// TIA Portal V15.1 export
// export: Created 2024-05-17T05:38:27.6005423Z, ExportSetting WithDefaults, DisplayName Totally Integrated Automation Portal, DisplayVersion V15.1 Update 5, DisplayName TIA Portal Openness, DisplayVersion V15.1 Update 5, DisplayName SINAMICS Startdrive Advanced, DisplayVersion V15.1, DisplayName G130, G150, S120, S150, SINAMICS MV, S210, DisplayVersion V15.1, DisplayName G110M, G120, G120C, G120D, G120P, DisplayVersion V15.1, DisplayName STEP 7 Professional, DisplayVersion V15.1 Update 5, DisplayName STEP 7 Safety, DisplayVersion V15.1, DisplayName WinCC Professional, DisplayVersion V15.1 Update 5, DisplayName SIMATIC Visualization Architect, DisplayVersion V15.1
FUNCTION "LETAFuseModule09_16_CPC20PN-Config" : Void   // FC1407, SCL
{ S7_Optimized_Access := 'TRUE' }
VERSION : 0.1
// stored: AutoNumber false, IsIECCheckEnabled false, SetENOAutomatically False, UDAEnableTagReadback false
   VAR_INPUT
      I_FuseMod9_Used : Bool;   // Fuse module is used
      I_FuseMod9_CH1_NominalCurrent : Int;   // Nominal current for the fuse
      I_FuseMod9_CH1_Name : String;   // Fuse name
      I_FuseMod9_CH1_Description : String;   // Description
      I_FuseMod9_CH2_NominalCurrent : Int;   // Nominal current for the fuse
      I_FuseMod9_CH2_Name : String;   // Fuse name
      I_FuseMod9_CH2_Description : String;   // Description
      I_FuseMod10_Used : Bool;   // Fuse module is used
      I_FuseMod10_CH1_NominalCurrent : Int;   // Nominal current for the fuse
      I_FuseMod10_CH1_Name : String;   // Fuse name
      I_FuseMod10_CH1_Description : String;   // Description
      I_FuseMod10_CH2_NominalCurrent : Int;   // Nominal current for the fuse
      I_FuseMod10_CH2_Name : String;   // Fuse name
      I_FuseMod10_CH2_Description : String;   // Description
      I_FuseMod11_Used : Bool;   // Fuse module is used
      I_FuseMod11_CH1_NominalCurrent : Int;   // Nominal current for the fuse
      I_FuseMod11_CH1_Name : String;   // Fuse name
      I_FuseMod11_CH1_Description : String;   // Description
      I_FuseMod11_CH2_NominalCurrent : Int;   // Nominal current for the fuse
      I_FuseMod11_CH2_Name : String;   // Fuse name
      I_FuseMod11_CH2_Description : String;   // Description
      I_FuseMod12_Used : Bool;   // Fuse module is used
      I_FuseMod12_CH1_NominalCurrent : Int;   // Nominal current for the fuse
      I_FuseMod12_CH1_Name : String;   // Fuse name
      I_FuseMod12_CH1_Description : String;   // Description
      I_FuseMod12_CH2_NominalCurrent : Int;   // Nominal current for the fuse
      I_FuseMod12_CH2_Name : String;   // Fuse name
      I_FuseMod12_CH2_Description : String;   // Description
      I_FuseMod13_Used : Bool;   // Fuse module is used
      I_FuseMod13_CH1_NominalCurrent : Int;   // Nominal current for the fuse
      I_FuseMod13_CH1_Name : String;   // Fuse name
      I_FuseMod13_CH1_Description : String;   // Description
      I_FuseMod13_CH2_NominalCurrent : Int;   // Nominal current for the fuse
      I_FuseMod13_CH2_Name : String;   // Fuse name
      I_FuseMod13_CH2_Description : String;   // Description
      I_FuseMod14_Used : Bool;   // Fuse module is used
      I_FuseMod14_CH1_NominalCurrent : Int;   // Nominal current for the fuse
      I_FuseMod14_CH1_Name : String;   // Fuse name
      I_FuseMod14_CH1_Description : String;   // Description
      I_FuseMod14_CH2_NominalCurrent : Int;   // Nominal current for the fuse
      I_FuseMod14_CH2_Name : String;   // Fuse name
      I_FuseMod14_CH2_Description : String;   // Description
      I_FuseMod15_Used : Bool;   // Fuse module is used
      I_FuseMod15_CH1_NominalCurrent : Int;   // Nominal current for the fuse
      I_FuseMod15_CH1_Name : String;   // Fuse name
      I_FuseMod15_CH1_Description : String;   // Description
      I_FuseMod15_CH2_NominalCurrent : Int;   // Nominal current for the fuse
      I_FuseMod15_CH2_Name : String;   // Fuse name
      I_FuseMod15_CH2_Description : String;   // Description
      I_FuseMod16_Used : Bool;   // Fuse module is used
      I_FuseMod16_CH1_NominalCurrent : Int;   // Nominal current for the fuse
      I_FuseMod16_CH1_Name : String;   // Fuse name
      I_FuseMod16_CH1_Description : String;   // Description
      I_FuseMod16_CH2_NominalCurrent : Int;   // Nominal current for the fuse
      I_FuseMod16_CH2_Name : String;   // Fuse name
      I_FuseMod16_CH2_Description : String;   // Description
   END_VAR
   VAR_IN_OUT
      IO_Config : "ETAFuseCPC20PNConfig";
   END_VAR
BEGIN
   #IO_Config.Fuse[17].Used := #I_FuseMod9_Used;
   #IO_Config.Fuse[17].NominalCurrent := #I_FuseMod9_CH1_NominalCurrent;
   #IO_Config.Fuse[17].Name := #I_FuseMod9_CH1_Name;
   #IO_Config.Fuse[17].Description := #I_FuseMod9_CH1_Description;

   #IO_Config.Fuse[18].Used := #I_FuseMod9_Used;
   #IO_Config.Fuse[18].NominalCurrent := #I_FuseMod9_CH2_NominalCurrent;
   #IO_Config.Fuse[18].Name := #I_FuseMod9_CH2_Name;
   #IO_Config.Fuse[18].Description := #I_FuseMod9_CH2_Description;

   #IO_Config.Fuse[19].Used := #I_FuseMod10_Used;
   #IO_Config.Fuse[19].NominalCurrent := #I_FuseMod10_CH1_NominalCurrent;
   #IO_Config.Fuse[19].Name := #I_FuseMod10_CH1_Name;
   #IO_Config.Fuse[19].Description := #I_FuseMod10_CH1_Description;

   #IO_Config.Fuse[20].Used := #I_FuseMod10_Used;
   #IO_Config.Fuse[20].NominalCurrent := #I_FuseMod10_CH2_NominalCurrent;
   #IO_Config.Fuse[20].Name := #I_FuseMod10_CH2_Name;
   #IO_Config.Fuse[20].Description := #I_FuseMod10_CH2_Description;

   #IO_Config.Fuse[21].Used := #I_FuseMod11_Used;
   #IO_Config.Fuse[21].NominalCurrent := #I_FuseMod11_CH1_NominalCurrent;
   #IO_Config.Fuse[21].Name := #I_FuseMod11_CH1_Name;
   #IO_Config.Fuse[21].Description := #I_FuseMod11_CH1_Description;

   #IO_Config.Fuse[22].Used := #I_FuseMod11_Used;
   #IO_Config.Fuse[22].NominalCurrent := #I_FuseMod11_CH2_NominalCurrent;
   #IO_Config.Fuse[22].Name := #I_FuseMod11_CH2_Name;
   #IO_Config.Fuse[22].Description := #I_FuseMod11_CH2_Description;

   #IO_Config.Fuse[23].Used := #I_FuseMod12_Used;
   #IO_Config.Fuse[23].NominalCurrent := #I_FuseMod12_CH1_NominalCurrent;
   #IO_Config.Fuse[23].Name := #I_FuseMod12_CH1_Name;
   #IO_Config.Fuse[23].Description := #I_FuseMod12_CH1_Description;

   #IO_Config.Fuse[24].Used := #I_FuseMod12_Used;
   #IO_Config.Fuse[24].NominalCurrent := #I_FuseMod12_CH2_NominalCurrent;
   #IO_Config.Fuse[24].Name := #I_FuseMod12_CH2_Name;
   #IO_Config.Fuse[24].Description := #I_FuseMod12_CH2_Description;

   #IO_Config.Fuse[25].Used := #I_FuseMod13_Used;
   #IO_Config.Fuse[25].NominalCurrent := #I_FuseMod13_CH1_NominalCurrent;
   #IO_Config.Fuse[25].Name := #I_FuseMod13_CH1_Name;
   #IO_Config.Fuse[25].Description := #I_FuseMod13_CH1_Description;

   #IO_Config.Fuse[26].Used := #I_FuseMod13_Used;
   #IO_Config.Fuse[26].NominalCurrent := #I_FuseMod13_CH2_NominalCurrent;
   #IO_Config.Fuse[26].Name := #I_FuseMod13_CH2_Name;
   #IO_Config.Fuse[26].Description := #I_FuseMod13_CH2_Description;

   #IO_Config.Fuse[27].Used := #I_FuseMod14_Used;
   #IO_Config.Fuse[27].NominalCurrent := #I_FuseMod14_CH1_NominalCurrent;
   #IO_Config.Fuse[27].Name := #I_FuseMod14_CH1_Name;
   #IO_Config.Fuse[27].Description := #I_FuseMod14_CH1_Description;

   #IO_Config.Fuse[28].Used := #I_FuseMod14_Used;
   #IO_Config.Fuse[28].NominalCurrent := #I_FuseMod14_CH2_NominalCurrent;
   #IO_Config.Fuse[28].Name := #I_FuseMod14_CH2_Name;
   #IO_Config.Fuse[28].Description := #I_FuseMod14_CH2_Description;

   #IO_Config.Fuse[29].Used := #I_FuseMod15_Used;
   #IO_Config.Fuse[29].NominalCurrent := #I_FuseMod15_CH1_NominalCurrent;
   #IO_Config.Fuse[29].Name := #I_FuseMod15_CH1_Name;
   #IO_Config.Fuse[29].Description := #I_FuseMod15_CH1_Description;

   #IO_Config.Fuse[30].Used := #I_FuseMod15_Used;
   #IO_Config.Fuse[30].NominalCurrent := #I_FuseMod15_CH2_NominalCurrent;
   #IO_Config.Fuse[30].Name := #I_FuseMod15_CH2_Name;
   #IO_Config.Fuse[30].Description := #I_FuseMod15_CH2_Description;

   #IO_Config.Fuse[31].Used := #I_FuseMod16_Used;
   #IO_Config.Fuse[31].NominalCurrent := #I_FuseMod16_CH1_NominalCurrent;
   #IO_Config.Fuse[31].Name := #I_FuseMod16_CH1_Name;
   #IO_Config.Fuse[31].Description := #I_FuseMod16_CH1_Description;

   #IO_Config.Fuse[32].Used := #I_FuseMod16_Used;
   #IO_Config.Fuse[32].NominalCurrent := #I_FuseMod16_CH2_NominalCurrent;
   #IO_Config.Fuse[32].Name := #I_FuseMod16_CH2_Name;
   #IO_Config.Fuse[32].Description := #I_FuseMod16_CH2_Description;
END_FUNCTION
